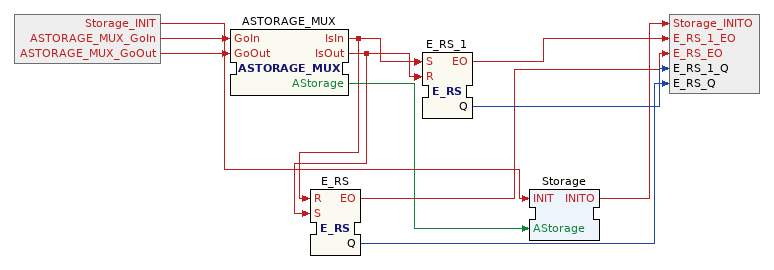
      [picture p48: application VDMA_Station1_HierarchicalControl_Distributed.StorageInternalLogicSubApp]
      FBS
        ASTORAGE_MUX : ASTORAGE_MUX;
        E_RS_1 : E_RS;
        E_RS : E_RS;
      END_FBS
      SUBAPPLICATION Storage
        EVENT_INPUT
          INIT;
        END_EVENT
        EVENT_OUTPUT
          INITO;
        END_EVENT
        SOCKETS
          AStorage : AStorage;
        END_SOCKETS
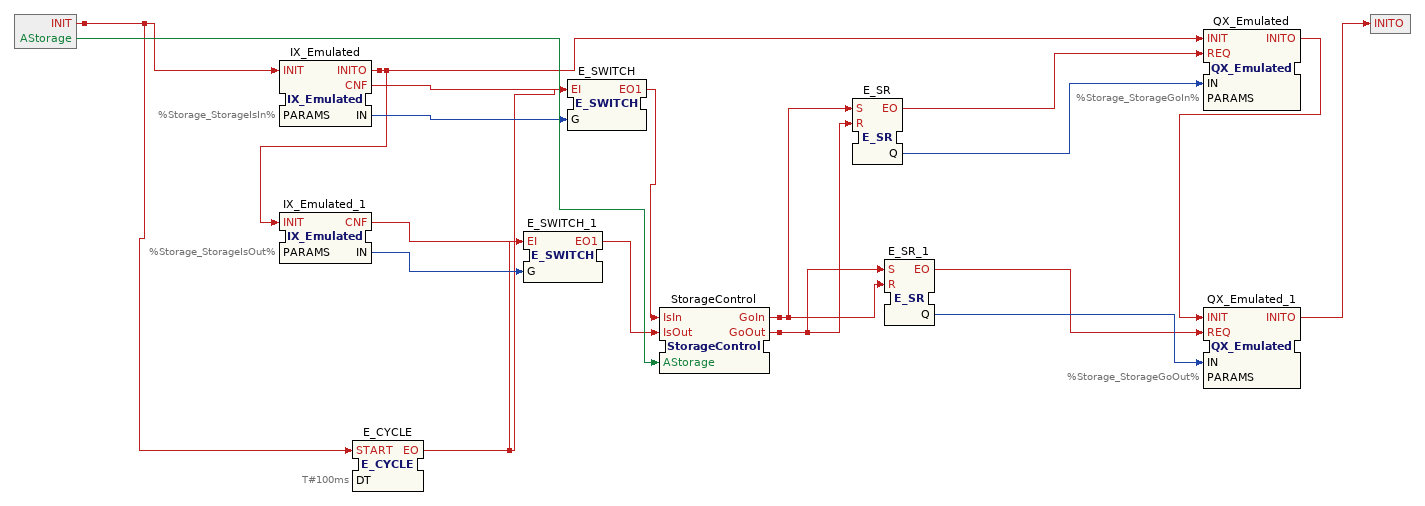
        FBS
          IX_Emulated : IX_Emulated(PARAMS := %Storage_StorageIsIn%);
          E_SWITCH : E_SWITCH;
          E_SR : E_SR;
          E_SR_1 : E_SR;
          StorageControl : StorageControl;
          E_SWITCH_1 : E_SWITCH;
          IX_Emulated_1 : IX_Emulated(PARAMS := %Storage_StorageIsOut%);
          E_CYCLE : E_CYCLE(DT := T#100ms);
          QX_Emulated_1 : QX_Emulated(PARAMS := %Storage_StorageGoOut%);
          QX_Emulated : QX_Emulated(PARAMS := %Storage_StorageGoIn%);
        END_FBS
        EVENT_CONNECTIONS
          IX_Emulated.INITO TO IX_Emulated_1.INIT;
          IX_Emulated.CNF TO E_SWITCH.EI;
          E_SWITCH.EO1 TO StorageControl.IsIn;
          StorageControl.GoIn TO E_SR.S;
          StorageControl.GoOut TO E_SR.R;
          StorageControl.GoOut TO E_SR_1.S;
          StorageControl.GoIn TO E_SR_1.R;
          E_SWITCH_1.EO1 TO StorageControl.IsOut;
          IX_Emulated_1.CNF TO E_SWITCH_1.EI;
          INIT TO IX_Emulated.INIT;
          INIT TO E_CYCLE.START;
          QX_Emulated_1.INITO TO INITO;
          IX_Emulated.INITO TO QX_Emulated.INIT;
          QX_Emulated.INITO TO QX_Emulated_1.INIT;
          E_SR.EO TO QX_Emulated.REQ;
          E_SR_1.EO TO QX_Emulated_1.REQ;
          E_CYCLE.EO TO E_SWITCH.EI;
          E_CYCLE.EO TO E_SWITCH_1.EI;
        END_CONNECTIONS
        DATA_CONNECTIONS
          IX_Emulated.IN TO E_SWITCH.G;
          IX_Emulated_1.IN TO E_SWITCH_1.G;
          E_SR.Q TO QX_Emulated.IN;
          E_SR_1.Q TO QX_Emulated_1.IN;
        END_CONNECTIONS
        ADAPTER_CONNECTIONS
          AStorage TO StorageControl.AStorage;
        END_CONNECTIONS
      END_SUBAPPLICATION
      EVENT_CONNECTIONS
        ASTORAGE_MUX.IsIn TO E_RS.R;
        ASTORAGE_MUX.IsIn TO E_RS_1.S;
        ASTORAGE_MUX.IsOut TO E_RS.S;
        ASTORAGE_MUX.IsOut TO E_RS_1.R;
        Storage_INIT TO Storage.INIT;
        Storage.INITO TO Storage_INITO;
        ASTORAGE_MUX_GoIn TO ASTORAGE_MUX.GoIn;
        ASTORAGE_MUX_GoOut TO ASTORAGE_MUX.GoOut;
        E_RS_1.EO TO E_RS_1_EO;
        E_RS.EO TO E_RS_EO;
      END_CONNECTIONS
      DATA_CONNECTIONS
        E_RS_1.Q TO E_RS_1_Q;
        E_RS.Q TO E_RS_Q;
      END_CONNECTIONS
      ADAPTER_CONNECTIONS
        ASTORAGE_MUX.AStorage TO Storage.AStorage;
      END_CONNECTIONS
    END_SUBAPPLICATION
    SUBAPPLICATION TurntableInternalLogicSubApp
      EVENT_INPUT
        ATURNTABLE_MUX_NewPosition;
        Turntable_INIT;
      END_EVENT
      EVENT_OUTPUT
        ATURNTABLE_MUX_PositionUpd;
        Turntable_INITO;
      END_EVENT
      VAR_INPUT
        ATURNTABLE_MUX_Position : WORD;
      END_VAR
      VAR_OUTPUT
        ATURNTABLE_MUX_CurrentPosition : WORD;
      END_VAR
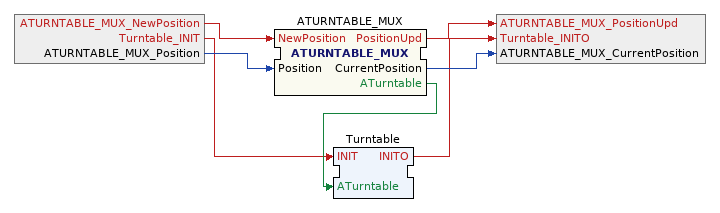
      FBS
        ATURNTABLE_MUX : ATURNTABLE_MUX;
      END_FBS
      SUBAPPLICATION Turntable
        EVENT_INPUT
          INIT;
        END_EVENT
        EVENT_OUTPUT
          INITO;
        END_EVENT
        SOCKETS
          ATurntable : ATurntable;
        END_SOCKETS
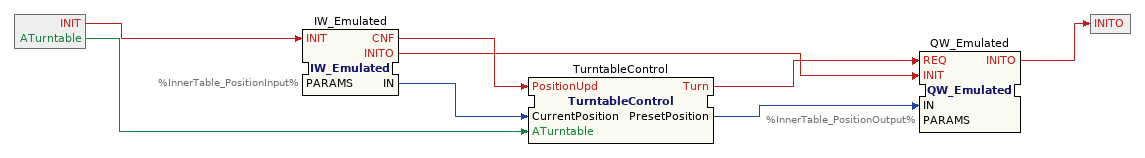
        FBS
          QW_Emulated : QW_Emulated(PARAMS := %InnerTable_PositionOutput%);
          IW_Emulated : IW_Emulated(PARAMS := %InnerTable_PositionInput%);
          TurntableControl : TurntableControl;
        END_FBS
        EVENT_CONNECTIONS
          TurntableControl.Turn TO QW_Emulated.REQ;
          IW_Emulated.CNF TO TurntableControl.PositionUpd;
          IW_Emulated.INITO TO QW_Emulated.INIT;
          INIT TO IW_Emulated.INIT;
          QW_Emulated.INITO TO INITO;
        END_CONNECTIONS
        DATA_CONNECTIONS
          TurntableControl.PresetPosition TO QW_Emulated.IN;
          IW_Emulated.IN TO TurntableControl.CurrentPosition;
        END_CONNECTIONS
        ADAPTER_CONNECTIONS
          ATurntable TO TurntableControl.ATurntable;
        END_CONNECTIONS
      END_SUBAPPLICATION
      EVENT_CONNECTIONS
        ATURNTABLE_MUX_NewPosition TO ATURNTABLE_MUX.NewPosition;
        ATURNTABLE_MUX.PositionUpd TO ATURNTABLE_MUX_PositionUpd;
        Turntable_INIT TO Turntable.INIT;
        Turntable.INITO TO Turntable_INITO;
      END_CONNECTIONS
      DATA_CONNECTIONS
        ATURNTABLE_MUX_Position TO ATURNTABLE_MUX.Position;
        ATURNTABLE_MUX.CurrentPosition TO ATURNTABLE_MUX_CurrentPosition;
      END_CONNECTIONS
      ADAPTER_CONNECTIONS
        ATURNTABLE_MUX.ATurntable TO Turntable.ATurntable;
      END_CONNECTIONS
    END_SUBAPPLICATION
    SUBAPPLICATION GripperInternalLogicSubApp
      EVENT_INPUT
        Gripper_INIT;
        AGRIPPER_MUX_Grip;
        AGRIPPER_MUX_Release;
      END_EVENT
      EVENT_OUTPUT
        E_RS_3_EO;
        Gripper_INITO;
        E_RS_2_EO;
      END_EVENT
      VAR_OUTPUT
        E_RS_3_Q : BOOL;
        E_RS_2_Q : BOOL;
      END_VAR
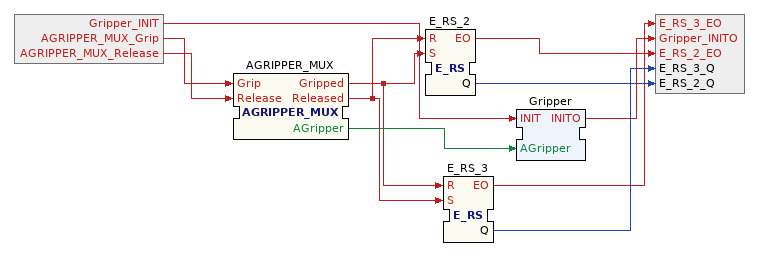
      FBS
        E_RS_3 : E_RS;
        E_RS_2 : E_RS;
        AGRIPPER_MUX : AGRIPPER_MUX;
      END_FBS
      SUBAPPLICATION Gripper
        EVENT_INPUT
          INIT;
        END_EVENT
        EVENT_OUTPUT
          INITO;
        END_EVENT
        SOCKETS
          AGripper : AGripper;
        END_SOCKETS
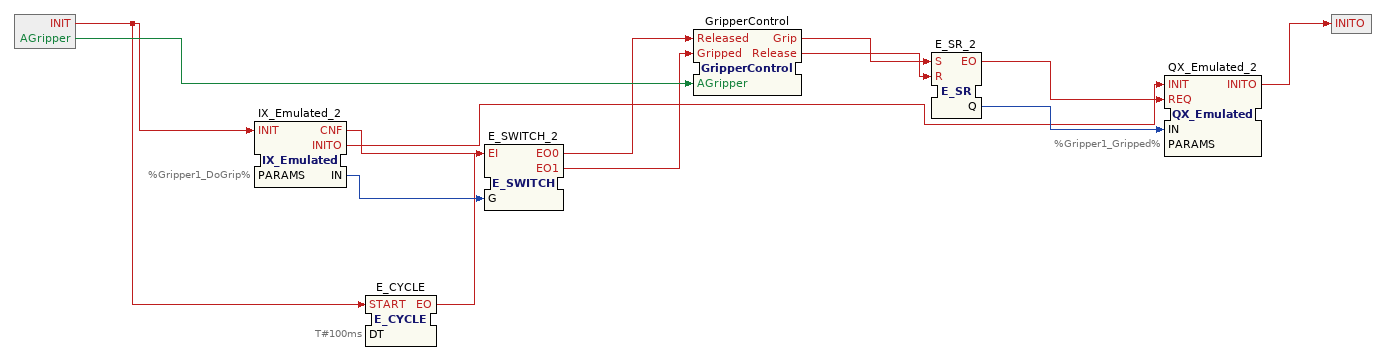
        FBS
          IX_Emulated_2 : IX_Emulated(PARAMS := %Gripper1_DoGrip%);
          E_SWITCH_2 : E_SWITCH;
          GripperControl : GripperControl;
          E_SR_2 : E_SR;
          E_CYCLE : E_CYCLE(DT := T#100ms);
          QX_Emulated_2 : QX_Emulated(PARAMS := %Gripper1_Gripped%);
        END_FBS
        EVENT_CONNECTIONS
          IX_Emulated_2.CNF TO E_SWITCH_2.EI;
          E_SWITCH_2.EO0 TO GripperControl.Released;
          E_SWITCH_2.EO1 TO GripperControl.Gripped;
          GripperControl.Grip TO E_SR_2.S;
          GripperControl.Release TO E_SR_2.R;
          E_CYCLE.EO TO E_SWITCH_2.EI;
          INIT TO E_CYCLE.START;
          INIT TO IX_Emulated_2.INIT;
          IX_Emulated_2.INITO TO QX_Emulated_2.INIT;
          QX_Emulated_2.INITO TO INITO;
          E_SR_2.EO TO QX_Emulated_2.REQ;
        END_CONNECTIONS
        DATA_CONNECTIONS
          IX_Emulated_2.IN TO E_SWITCH_2.G;
          E_SR_2.Q TO QX_Emulated_2.IN;
        END_CONNECTIONS
        ADAPTER_CONNECTIONS
          AGripper TO GripperControl.AGripper;
        END_CONNECTIONS
      END_SUBAPPLICATION
      EVENT_CONNECTIONS
        AGRIPPER_MUX.Gripped TO E_RS_3.R;
        AGRIPPER_MUX.Released TO E_RS_3.S;
        AGRIPPER_MUX.Released TO E_RS_2.R;
        AGRIPPER_MUX.Gripped TO E_RS_2.S;
        E_RS_3.EO TO E_RS_3_EO;
        Gripper_INIT TO Gripper.INIT;
        Gripper.INITO TO Gripper_INITO;
        E_RS_2.EO TO E_RS_2_EO;
        AGRIPPER_MUX_Grip TO AGRIPPER_MUX.Grip;
        AGRIPPER_MUX_Release TO AGRIPPER_MUX.Release;
      END_CONNECTIONS
      DATA_CONNECTIONS
        E_RS_3.Q TO E_RS_3_Q;
        E_RS_2.Q TO E_RS_2_Q;
      END_CONNECTIONS
      ADAPTER_CONNECTIONS
        AGRIPPER_MUX.AGripper TO Gripper.AGripper;
      END_CONNECTIONS
    END_SUBAPPLICATION
    SUBAPPLICATION RobotInternalLogicSubApp
      EVENT_INPUT
        AROBOT_MUX_PresetPositionUpd;
        Robot_INIT;
      END_EVENT
      EVENT_OUTPUT
        AROBOT_MUX_PositionUpdate;
        Robot_INITO;
      END_EVENT
      VAR_INPUT
        AROBOT_MUX_PresetPosition : WORD;
      END_VAR
      VAR_OUTPUT
        AROBOT_MUX_CurrentPosition : WORD;
      END_VAR
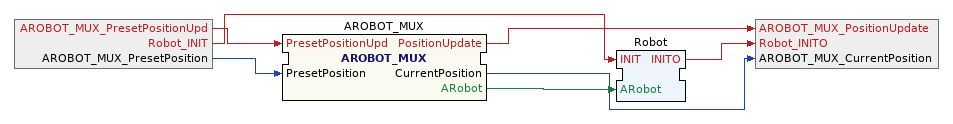
      FBS
        AROBOT_MUX : AROBOT_MUX;
      END_FBS
      SUBAPPLICATION Robot
        EVENT_INPUT
          INIT;
        END_EVENT
        EVENT_OUTPUT
          INITO;
        END_EVENT
        SOCKETS
          ARobot : ARobot;
        END_SOCKETS
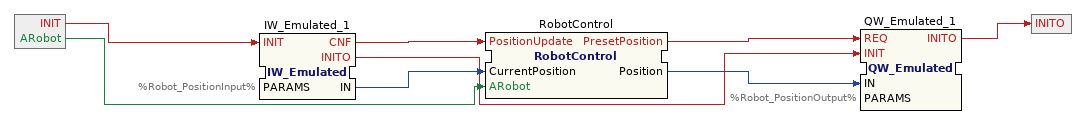
        FBS
          IW_Emulated_1 : IW_Emulated(PARAMS := %Robot_PositionInput%);
          RobotControl : RobotControl;
          QW_Emulated_1 : QW_Emulated(PARAMS := %Robot_PositionOutput%);
        END_FBS
        EVENT_CONNECTIONS
          IW_Emulated_1.CNF TO RobotControl.PositionUpdate;
          RobotControl.PresetPosition TO QW_Emulated_1.REQ;
          IW_Emulated_1.INITO TO QW_Emulated_1.INIT;
          QW_Emulated_1.INITO TO INITO;
          INIT TO IW_Emulated_1.INIT;
        END_CONNECTIONS
        DATA_CONNECTIONS
          IW_Emulated_1.IN TO RobotControl.CurrentPosition;
          RobotControl.Position TO QW_Emulated_1.IN;
        END_CONNECTIONS
        ADAPTER_CONNECTIONS
          ARobot TO RobotControl.ARobot;
        END_CONNECTIONS
      END_SUBAPPLICATION
      EVENT_CONNECTIONS
        AROBOT_MUX_PresetPositionUpd TO AROBOT_MUX.PresetPositionUpd;
        AROBOT_MUX.PositionUpdate TO AROBOT_MUX_PositionUpdate;
        Robot_INIT TO Robot.INIT;
        Robot.INITO TO Robot_INITO;
      END_CONNECTIONS
      DATA_CONNECTIONS
        AROBOT_MUX_PresetPosition TO AROBOT_MUX.PresetPosition;
        AROBOT_MUX.CurrentPosition TO AROBOT_MUX_CurrentPosition;
      END_CONNECTIONS
      ADAPTER_CONNECTIONS
        AROBOT_MUX.ARobot TO Robot.ARobot;
      END_CONNECTIONS
    END_SUBAPPLICATION
    EVENT_CONNECTIONS
      SERVER_0.IND TO SERVER_0.RSP;
      SERVER_1.IND TO SERVER_1.RSP;
      SERVER_0.INITO TO SERVER_1.INIT;
      SERVER_5.IND TO SERVER_5.RSP;
      SERVER_4.IND TO SERVER_4.RSP;
      SERVER_4.INITO TO SERVER_5.INIT;
      CLIENT_4.INITO TO CLIENT_5.INIT;
      CLIENT_0.INITO TO CLIENT_3.INIT;
      SUBSCRIBE_2.IND TO TurntableSubApp.PositionUpd;
      SUBSCRIBE_1.IND TO RobotSubApp.PositionUpdate;
      SERVER_5.INITO TO PUBLISH_5.INIT;
      PUBLISH_5.INITO TO PUBLISH_4.INIT;
      SUBSCRIBE_3.INITO TO CLIENT_0.INIT;
      SERVER_1.INITO TO PUBLISH_0.INIT;
      PUBLISH_0.INITO TO PUBLISH_1.INIT;
      SUBSCRIBE_2.INITO TO SUBSCRIBE_4.INIT;
      SUBSCRIBE_4.INITO TO SUBSCRIBE_5.INIT;
      SUBSCRIBE_5.INITO TO CLIENT_4.INIT;
      SUBSCRIBE_5.INITO TO SUBSCRIBE_1.INIT;
      SUBSCRIBE_9.INITO TO SUBSCRIBE_3.INIT;
      CLIENT_3.INITO TO SUBSCRIBE_2.INIT;
      SERVER_3.IND TO SERVER_3.RSP;
      SERVER_3.INITO TO PUBLISH_3.INIT;
      SUBSCRIBE_2.INITO TO CLIENT_2.INIT;
      TurntableSubApp.NewPosition TO CLIENT_2.REQ;
      SUBSCRIBE_1.INITO TO CLIENT_1.INIT;
      RobotSubApp.PresetPositionUpd TO CLIENT_1.REQ;
      SERVER_2.IND TO SERVER_2.RSP;
      SERVER_2.INITO TO PUBLISH_2.INIT;
      SUBSCRIBE_9.IND TO StorageSubApp.E_SWITCH_1_EI;
      SUBSCRIBE_3.IND TO StorageSubApp.E_SWITCH_EI;
      StorageSubApp.ASTORAGE_DEMUX_GoIn TO CLIENT_0.REQ;
      StorageSubApp.ASTORAGE_DEMUX_GoOut TO CLIENT_3.REQ;
      SUBSCRIBE_4.IND TO GripperSubApp.E_SWITCH_2_EI;
      GripperSubApp.AGRIPPER_DEMUX_Grip TO CLIENT_4.REQ;
      GripperSubApp.AGRIPPER_DEMUX_Release TO CLIENT_5.REQ;
      SUBSCRIBE_5.IND TO GripperSubApp.E_SWITCH_3_EI;
      SERVER_5.INITO TO StorageInternalLogicSubApp.Storage_INIT;
      SERVER_4.IND TO StorageInternalLogicSubApp.ASTORAGE_MUX_GoIn;
      SERVER_5.IND TO StorageInternalLogicSubApp.ASTORAGE_MUX_GoOut;
      StorageInternalLogicSubApp.E_RS_1_EO TO PUBLISH_5.REQ;
      StorageInternalLogicSubApp.E_RS_EO TO PUBLISH_4.REQ;
      SERVER_3.IND TO TurntableInternalLogicSubApp.ATURNTABLE_MUX_NewPosition;
      TurntableInternalLogicSubApp.ATURNTABLE_MUX_PositionUpd TO PUBLISH_3.REQ;
      StorageInternalLogicSubApp.Storage_INITO TO TurntableInternalLogicSubApp.Turntable_INIT;
      TurntableInternalLogicSubApp.Turntable_INITO TO SERVER_3.INIT;
      GripperInternalLogicSubApp.E_RS_3_EO TO PUBLISH_1.REQ;
      TurntableInternalLogicSubApp.Turntable_INITO TO GripperInternalLogicSubApp.Gripper_INIT;
      GripperInternalLogicSubApp.Gripper_INITO TO SERVER_0.INIT;
      GripperInternalLogicSubApp.E_RS_2_EO TO PUBLISH_0.REQ;
      SERVER_0.IND TO GripperInternalLogicSubApp.AGRIPPER_MUX_Grip;
      SERVER_1.IND TO GripperInternalLogicSubApp.AGRIPPER_MUX_Release;
      SERVER_2.IND TO RobotInternalLogicSubApp.AROBOT_MUX_PresetPositionUpd;
      RobotInternalLogicSubApp.AROBOT_MUX_PositionUpdate TO PUBLISH_2.REQ;
      GripperInternalLogicSubApp.Gripper_INITO TO RobotInternalLogicSubApp.Robot_INIT;
      RobotInternalLogicSubApp.Robot_INITO TO SERVER_2.INIT;
    END_CONNECTIONS
    DATA_CONNECTIONS
      SUBSCRIBE_1.RD_1 TO RobotSubApp.CurrentPosition;
      SUBSCRIBE_2.RD_1 TO TurntableSubApp.CurrentPosition;
      TurntableSubApp.Position TO CLIENT_2.SD_1;
      RobotSubApp.PresetPosition TO CLIENT_1.SD_1;
      SUBSCRIBE_9.RD_1 TO StorageSubApp.E_SWITCH_1_G;
      SUBSCRIBE_3.RD_1 TO StorageSubApp.E_SWITCH_G;
      SUBSCRIBE_4.RD_1 TO GripperSubApp.E_SWITCH_2_G;
      SUBSCRIBE_5.RD_1 TO GripperSubApp.E_SWITCH_3_G;
      StorageInternalLogicSubApp.E_RS_1_Q TO PUBLISH_5.SD_1;
      StorageInternalLogicSubApp.E_RS_Q TO PUBLISH_4.SD_1;
      SERVER_3.RD_1 TO TurntableInternalLogicSubApp.ATURNTABLE_MUX_Position;
      TurntableInternalLogicSubApp.ATURNTABLE_MUX_CurrentPosition TO PUBLISH_3.SD_1;
      GripperInternalLogicSubApp.E_RS_3_Q TO PUBLISH_1.SD_1;
      GripperInternalLogicSubApp.E_RS_2_Q TO PUBLISH_0.SD_1;
      SERVER_2.RD_1 TO RobotInternalLogicSubApp.AROBOT_MUX_PresetPosition;
      RobotInternalLogicSubApp.AROBOT_MUX_CurrentPosition TO PUBLISH_2.SD_1;
    END_CONNECTIONS
    ADAPTER_CONNECTIONS
      Station1Control.ADepot TO DepotControl.ADepot;
      Station1Control.AHandling TO HandlingControl.AHandling;
      HandlingControl.ARobot TO RobotSubApp.ARobot;
      DepotControl.ATurntable TO TurntableSubApp.ATurntable;
      DepotControl.AStorage TO StorageSubApp.ASTORAGE_DEMUX_AStorage;
      HandlingControl.AGripper TO GripperSubApp.AGRIPPER_DEMUX_AGripper;
    END_CONNECTIONS
  END_APPLICATION
  APPLICATION VDMA_Station1_SkillbasedControl_Distributed
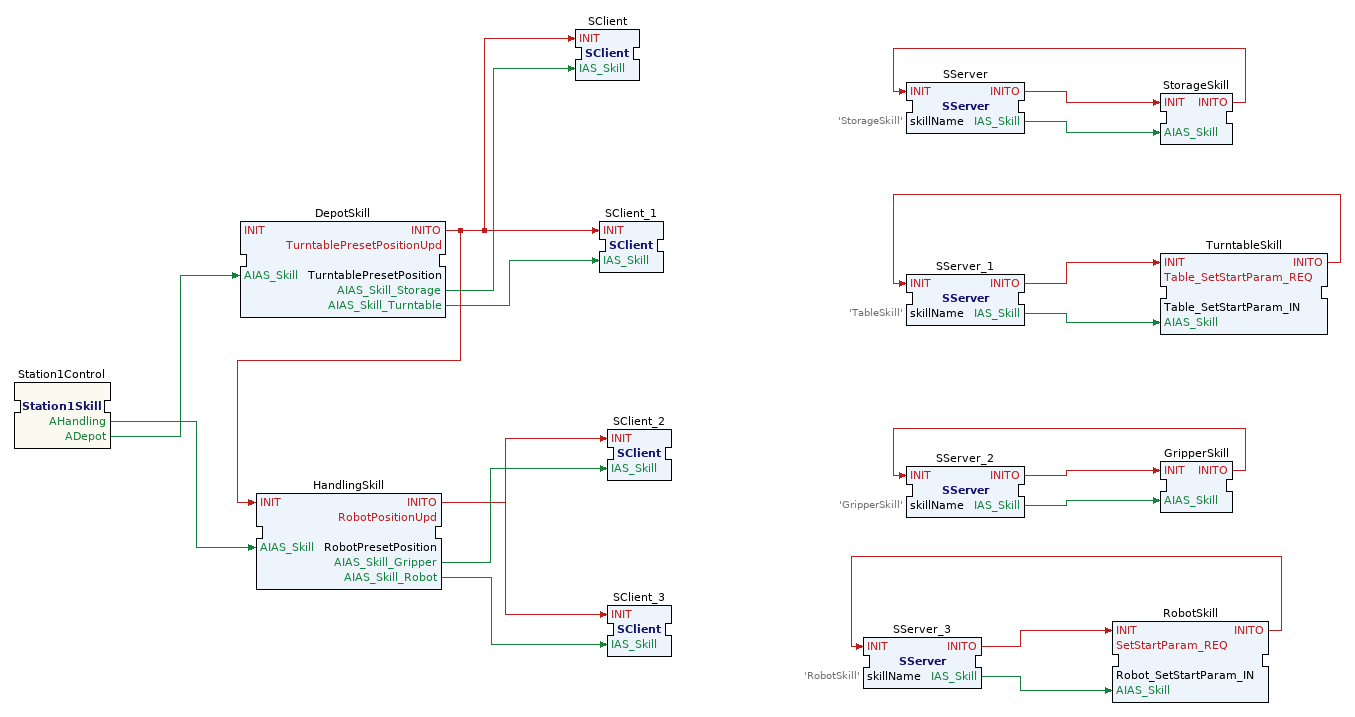
    FBS
      Station1Control : Station1Skill;
    END_FBS
    SUBAPPS
      SClient : SClient;
      SClient_1 : SClient;
      SClient_2 : SClient;
      SClient_3 : SClient;
      SServer : SServer(skillName := 'StorageSkill');
      SServer_1 : SServer(skillName := 'TableSkill');
      SServer_2 : SServer(skillName := 'GripperSkill');
      SServer_3 : SServer(skillName := 'RobotSkill');
    END_SUBAPPS
    SUBAPPLICATION StorageSkill
      EVENT_INPUT
        INIT;
      END_EVENT
      EVENT_OUTPUT
        INITO;
      END_EVENT
      SOCKETS
        AIAS_Skill : IAS_Skill;
      END_SOCKETS
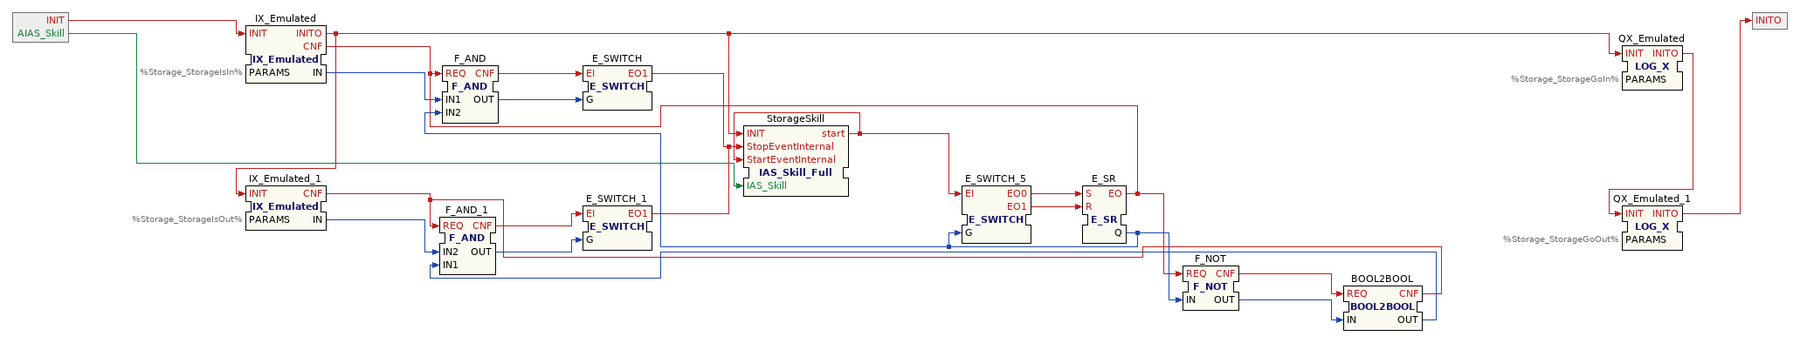
      FBS
        E_SWITCH_5 : E_SWITCH;
        IX_Emulated : IX_Emulated(PARAMS := %Storage_StorageIsIn%);
        QX_Emulated_1 : LOG_X(PARAMS := %Storage_StorageGoOut%);
        F_NOT : F_NOT;
        QX_Emulated : LOG_X(PARAMS := %Storage_StorageGoIn%);
        IX_Emulated_1 : IX_Emulated(PARAMS := %Storage_StorageIsOut%);
        E_SWITCH : E_SWITCH;
        E_SWITCH_1 : E_SWITCH;
        StorageSkill : IAS_Skill_Full;
        F_AND : F_AND;
        BOOL2BOOL : BOOL2BOOL;
        F_AND_1 : F_AND;
        E_SR : E_SR;
      END_FBS
      EVENT_CONNECTIONS
        StorageSkill.start TO E_SWITCH_5.EI;
        E_SWITCH_5.EO0 TO E_SR.S;
        E_SWITCH_5.EO1 TO E_SR.R;
        IX_Emulated.INITO TO IX_Emulated_1.INIT;
        IX_Emulated.INITO TO QX_Emulated.INIT;
        IX_Emulated.INITO TO StorageSkill.INIT;
        IX_Emulated.CNF TO F_AND.REQ;
        QX_Emulated.INITO TO QX_Emulated_1.INIT;
        E_SR.EO TO F_NOT.REQ;
        F_NOT.CNF TO BOOL2BOOL.REQ;
        IX_Emulated_1.CNF TO F_AND_1.REQ;
        F_AND.CNF TO E_SWITCH.EI;
        E_SWITCH.EO1 TO StorageSkill.StopEventInternal;
        F_AND_1.CNF TO E_SWITCH_1.EI;
        E_SWITCH_1.EO1 TO StorageSkill.StopEventInternal;
        StorageSkill.start TO StorageSkill.StartEventInternal;
        E_SR.EO TO F_AND.REQ;
        BOOL2BOOL.CNF TO F_AND_1.REQ;
        INIT TO IX_Emulated.INIT;
        QX_Emulated_1.INITO TO INITO;
      END_CONNECTIONS
      DATA_CONNECTIONS
        E_SR.Q TO E_SWITCH_5.G;
        IX_Emulated.IN TO F_AND.IN1;
        E_SR.Q TO F_NOT.IN;
        F_NOT.OUT TO BOOL2BOOL.IN;
        IX_Emulated_1.IN TO F_AND_1.IN2;
        F_AND.OUT TO E_SWITCH.G;
        F_AND_1.OUT TO E_SWITCH_1.G;
        E_SR.Q TO F_AND.IN2;
        BOOL2BOOL.OUT TO F_AND_1.IN1;
      END_CONNECTIONS
      ADAPTER_CONNECTIONS
        AIAS_Skill TO StorageSkill.IAS_Skill;
      END_CONNECTIONS
    END_SUBAPPLICATION
    SUBAPPLICATION TurntableSkill
      EVENT_INPUT
        INIT;
        Table_SetStartParam_REQ;
      END_EVENT
      EVENT_OUTPUT
        INITO;
      END_EVENT
      VAR_INPUT
        Table_SetStartParam_IN : WORD;
      END_VAR
      SOCKETS
        AIAS_Skill : IAS_Skill;
      END_SOCKETS
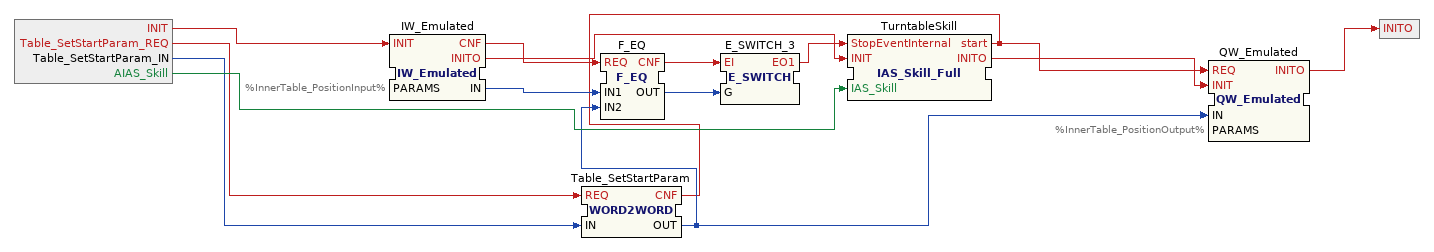
      FBS
        F_EQ : F_EQ;
        E_SWITCH_3 : E_SWITCH;
        Table_SetStartParam : WORD2WORD;
        QW_Emulated : QW_Emulated(PARAMS := %InnerTable_PositionOutput%);
        TurntableSkill : IAS_Skill_Full;
        IW_Emulated : IW_Emulated(PARAMS := %InnerTable_PositionInput%);
      END_FBS
      EVENT_CONNECTIONS
        IW_Emulated.CNF TO F_EQ.REQ;
        TurntableSkill.start TO F_EQ.REQ;
        Table_SetStartParam.CNF TO F_EQ.REQ;
        F_EQ.CNF TO E_SWITCH_3.EI;
        E_SWITCH_3.EO1 TO TurntableSkill.StopEventInternal;
        TurntableSkill.start TO QW_Emulated.REQ;
        Table_SetStartParam_REQ TO Table_SetStartParam.REQ;
        INIT TO IW_Emulated.INIT;
        IW_Emulated.INITO TO TurntableSkill.INIT;
        TurntableSkill.INITO TO QW_Emulated.INIT;
        QW_Emulated.INITO TO INITO;
      END_CONNECTIONS
      DATA_CONNECTIONS
        IW_Emulated.IN TO F_EQ.IN1;
        Table_SetStartParam.OUT TO F_EQ.IN2;
        F_EQ.OUT TO E_SWITCH_3.G;
        Table_SetStartParam.OUT TO QW_Emulated.IN;
        Table_SetStartParam_IN TO Table_SetStartParam.IN;
      END_CONNECTIONS
      ADAPTER_CONNECTIONS
        AIAS_Skill TO TurntableSkill.IAS_Skill;
      END_CONNECTIONS
    END_SUBAPPLICATION
    SUBAPPLICATION DepotSkill
      EVENT_INPUT
        INIT;
      END_EVENT
      EVENT_OUTPUT
        INITO;
        TurntablePresetPositionUpd;
      END_EVENT
      VAR_OUTPUT
        TurntablePresetPosition : WORD;
      END_VAR
      SOCKETS
        AIAS_Skill : IAS_Skill;
      END_SOCKETS
      PLUGS
        AIAS_Skill_Storage : IAS_Skill;
        AIAS_Skill_Turntable : IAS_Skill;
      END_PLUGS
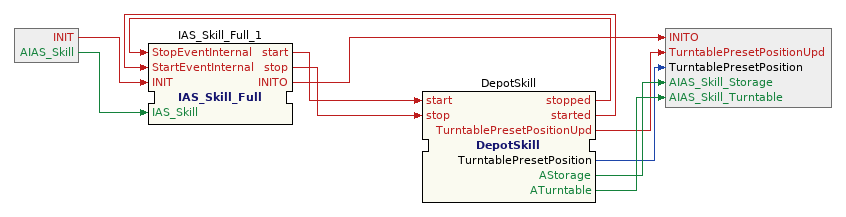
      FBS
        IAS_Skill_Full_1 : IAS_Skill_Full;
        DepotSkill : DepotSkill;
      END_FBS
      EVENT_CONNECTIONS
        DepotSkill.stopped TO IAS_Skill_Full_1.StopEventInternal;
        DepotSkill.started TO IAS_Skill_Full_1.StartEventInternal;
        IAS_Skill_Full_1.start TO DepotSkill.start;
        IAS_Skill_Full_1.stop TO DepotSkill.stop;
        DepotSkill.TurntablePresetPositionUpd TO TurntablePresetPositionUpd;
        INIT TO IAS_Skill_Full_1.INIT;
        IAS_Skill_Full_1.INITO TO INITO;
      END_CONNECTIONS
      DATA_CONNECTIONS
        DepotSkill.TurntablePresetPosition TO TurntablePresetPosition;
      END_CONNECTIONS
      ADAPTER_CONNECTIONS
        AIAS_Skill TO IAS_Skill_Full_1.IAS_Skill;
        DepotSkill.AStorage TO AIAS_Skill_Storage;
        DepotSkill.ATurntable TO AIAS_Skill_Turntable;
      END_CONNECTIONS
    END_SUBAPPLICATION
    SUBAPPLICATION GripperSkill
      EVENT_INPUT
        INIT;
      END_EVENT
      EVENT_OUTPUT
        INITO;
      END_EVENT
      SOCKETS
        AIAS_Skill : IAS_Skill;
      END_SOCKETS
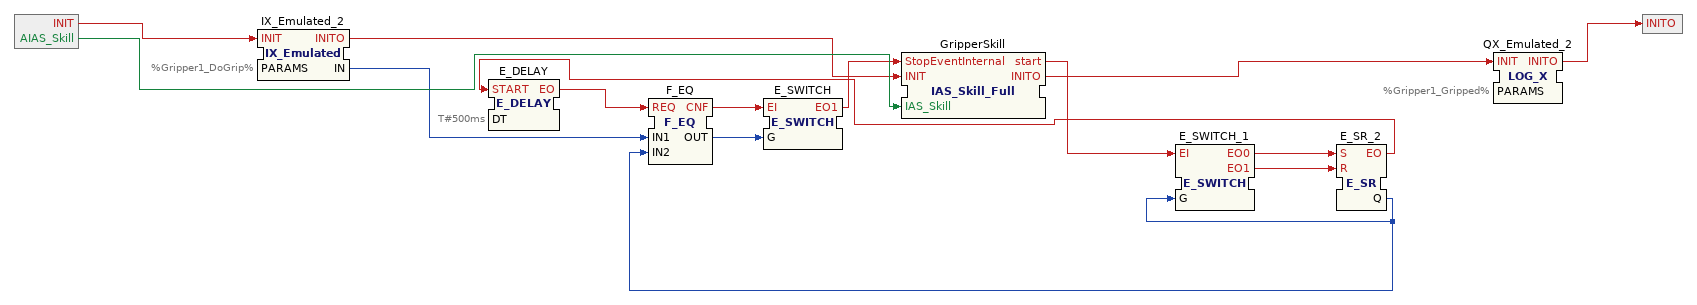
      FBS
        GripperSkill : IAS_Skill_Full;
        F_EQ : F_EQ;
        E_SWITCH_1 : E_SWITCH;
        IX_Emulated_2 : IX_Emulated(PARAMS := %Gripper1_DoGrip%);
        QX_Emulated_2 : LOG_X(PARAMS := %Gripper1_Gripped%);
        E_DELAY : E_DELAY(DT := T#500ms);
        E_SWITCH : E_SWITCH;
        E_SR_2 : E_SR;
      END_FBS
      EVENT_CONNECTIONS
        E_SWITCH.EO1 TO GripperSkill.StopEventInternal;
        GripperSkill.start TO E_SWITCH_1.EI;
        E_DELAY.EO TO F_EQ.REQ;
        F_EQ.CNF TO E_SWITCH.EI;
        E_SWITCH_1.EO0 TO E_SR_2.S;
        E_SWITCH_1.EO1 TO E_SR_2.R;
        E_SR_2.EO TO E_DELAY.START;
        INIT TO IX_Emulated_2.INIT;
        IX_Emulated_2.INITO TO GripperSkill.INIT;
        GripperSkill.INITO TO QX_Emulated_2.INIT;
        QX_Emulated_2.INITO TO INITO;
      END_CONNECTIONS
      DATA_CONNECTIONS
        IX_Emulated_2.IN TO F_EQ.IN1;
        E_SR_2.Q TO F_EQ.IN2;
        F_EQ.OUT TO E_SWITCH.G;
        E_SR_2.Q TO E_SWITCH_1.G;
      END_CONNECTIONS
      ADAPTER_CONNECTIONS
        AIAS_Skill TO GripperSkill.IAS_Skill;
      END_CONNECTIONS
    END_SUBAPPLICATION
    SUBAPPLICATION RobotSkill
      EVENT_INPUT
        INIT;
        SetStartParam_REQ;
      END_EVENT
      EVENT_OUTPUT
        INITO;
      END_EVENT
      VAR_INPUT
        Robot_SetStartParam_IN : WORD;
      END_VAR
      SOCKETS
        AIAS_Skill : IAS_Skill;
      END_SOCKETS
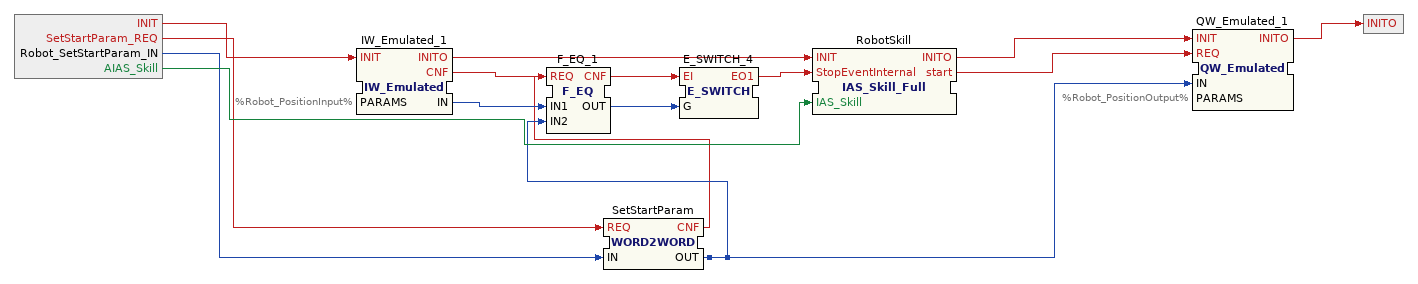
      FBS
        RobotSkill : IAS_Skill_Full;
        IW_Emulated_1 : IW_Emulated(PARAMS := %Robot_PositionInput%);
        E_SWITCH_4 : E_SWITCH;
        F_EQ_1 : F_EQ;
        QW_Emulated_1 : QW_Emulated(PARAMS := %Robot_PositionOutput%);
        SetStartParam : WORD2WORD;
      END_FBS
      EVENT_CONNECTIONS
        IW_Emulated_1.INITO TO RobotSkill.INIT;
        E_SWITCH_4.EO1 TO RobotSkill.StopEventInternal;
        RobotSkill.INITO TO QW_Emulated_1.INIT;
        RobotSkill.start TO QW_Emulated_1.REQ;
        IW_Emulated_1.CNF TO F_EQ_1.REQ;
        F_EQ_1.CNF TO E_SWITCH_4.EI;
        SetStartParam.CNF TO F_EQ_1.REQ;
        INIT TO IW_Emulated_1.INIT;
        SetStartParam_REQ TO SetStartParam.REQ;
        QW_Emulated_1.INITO TO INITO;
      END_CONNECTIONS
      DATA_CONNECTIONS
        IW_Emulated_1.IN TO F_EQ_1.IN1;
        F_EQ_1.OUT TO E_SWITCH_4.G;
        SetStartParam.OUT TO F_EQ_1.IN2;
        SetStartParam.OUT TO QW_Emulated_1.IN;
        Robot_SetStartParam_IN TO SetStartParam.IN;
      END_CONNECTIONS
      ADAPTER_CONNECTIONS
        AIAS_Skill TO RobotSkill.IAS_Skill;
      END_CONNECTIONS
    END_SUBAPPLICATION
    SUBAPPLICATION HandlingSkill
      EVENT_INPUT
        INIT;
      END_EVENT
      EVENT_OUTPUT
        INITO;
        RobotPositionUpd;
      END_EVENT
      VAR_OUTPUT
        RobotPresetPosition : WORD;
      END_VAR
      SOCKETS
        AIAS_Skill : IAS_Skill;
      END_SOCKETS
      PLUGS
        AIAS_Skill_Gripper : IAS_Skill;
        AIAS_Skill_Robot : IAS_Skill;
      END_PLUGS
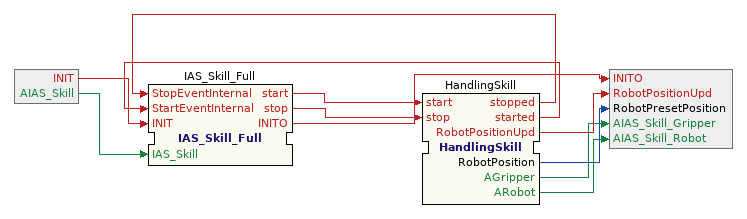
      FBS
        IAS_Skill_Full : IAS_Skill_Full;
        HandlingSkill : HandlingSkill;
      END_FBS
      EVENT_CONNECTIONS
        HandlingSkill.stopped TO IAS_Skill_Full.StopEventInternal;
        HandlingSkill.started TO IAS_Skill_Full.StartEventInternal;
        IAS_Skill_Full.start TO HandlingSkill.start;
        IAS_Skill_Full.stop TO HandlingSkill.stop;
        HandlingSkill.RobotPositionUpd TO RobotPositionUpd;
        INIT TO IAS_Skill_Full.INIT;
        IAS_Skill_Full.INITO TO INITO;
      END_CONNECTIONS
      DATA_CONNECTIONS
        HandlingSkill.RobotPosition TO RobotPresetPosition;
      END_CONNECTIONS
      ADAPTER_CONNECTIONS
        AIAS_Skill TO IAS_Skill_Full.IAS_Skill;
        HandlingSkill.AGripper TO AIAS_Skill_Gripper;
        HandlingSkill.ARobot TO AIAS_Skill_Robot;
      END_CONNECTIONS
    END_SUBAPPLICATION
    EVENT_CONNECTIONS
      DepotSkill.INITO TO HandlingSkill.INIT;
      HandlingSkill.INITO TO SClient_3.INIT;
      HandlingSkill.INITO TO SClient_2.INIT;
      DepotSkill.INITO TO SClient_1.INIT;
      DepotSkill.INITO TO SClient.INIT;
      SServer.INITO TO StorageSkill.INIT;
      StorageSkill.INITO TO SServer.INIT;
      SServer_1.INITO TO TurntableSkill.INIT;
      TurntableSkill.INITO TO SServer_1.INIT;
      SServer_2.INITO TO GripperSkill.INIT;
      GripperSkill.INITO TO SServer_2.INIT;
      SServer_3.INITO TO RobotSkill.INIT;
      RobotSkill.INITO TO SServer_3.INIT;
    END_CONNECTIONS
    ADAPTER_CONNECTIONS
      Station1Control.AHandling TO HandlingSkill.AIAS_Skill;
      Station1Control.ADepot TO DepotSkill.AIAS_Skill;
      DepotSkill.AIAS_Skill_Storage TO SClient.IAS_Skill;
      DepotSkill.AIAS_Skill_Turntable TO SClient_1.IAS_Skill;
      HandlingSkill.AIAS_Skill_Gripper TO SClient_2.IAS_Skill;
      HandlingSkill.AIAS_Skill_Robot TO SClient_3.IAS_Skill;
      SServer.IAS_Skill TO StorageSkill.AIAS_Skill;
      SServer_1.IAS_Skill TO TurntableSkill.AIAS_Skill;
      SServer_2.IAS_Skill TO GripperSkill.AIAS_Skill;
      SServer_3.IAS_Skill TO RobotSkill.AIAS_Skill;
    END_CONNECTIONS
  END_APPLICATION
  APPLICATION VDMA_Station1_EmulatorApp_SingleDevice
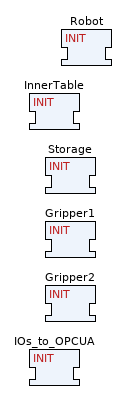
    SUBAPPLICATION Robot
      EVENT_INPUT
        INIT;
      END_EVENT
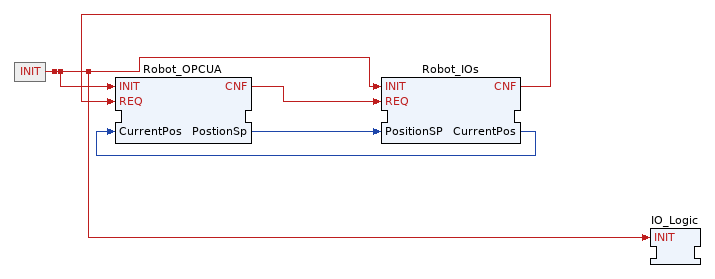
      SUBAPPLICATION IO_Logic
        EVENT_INPUT
          INIT;
        END_EVENT
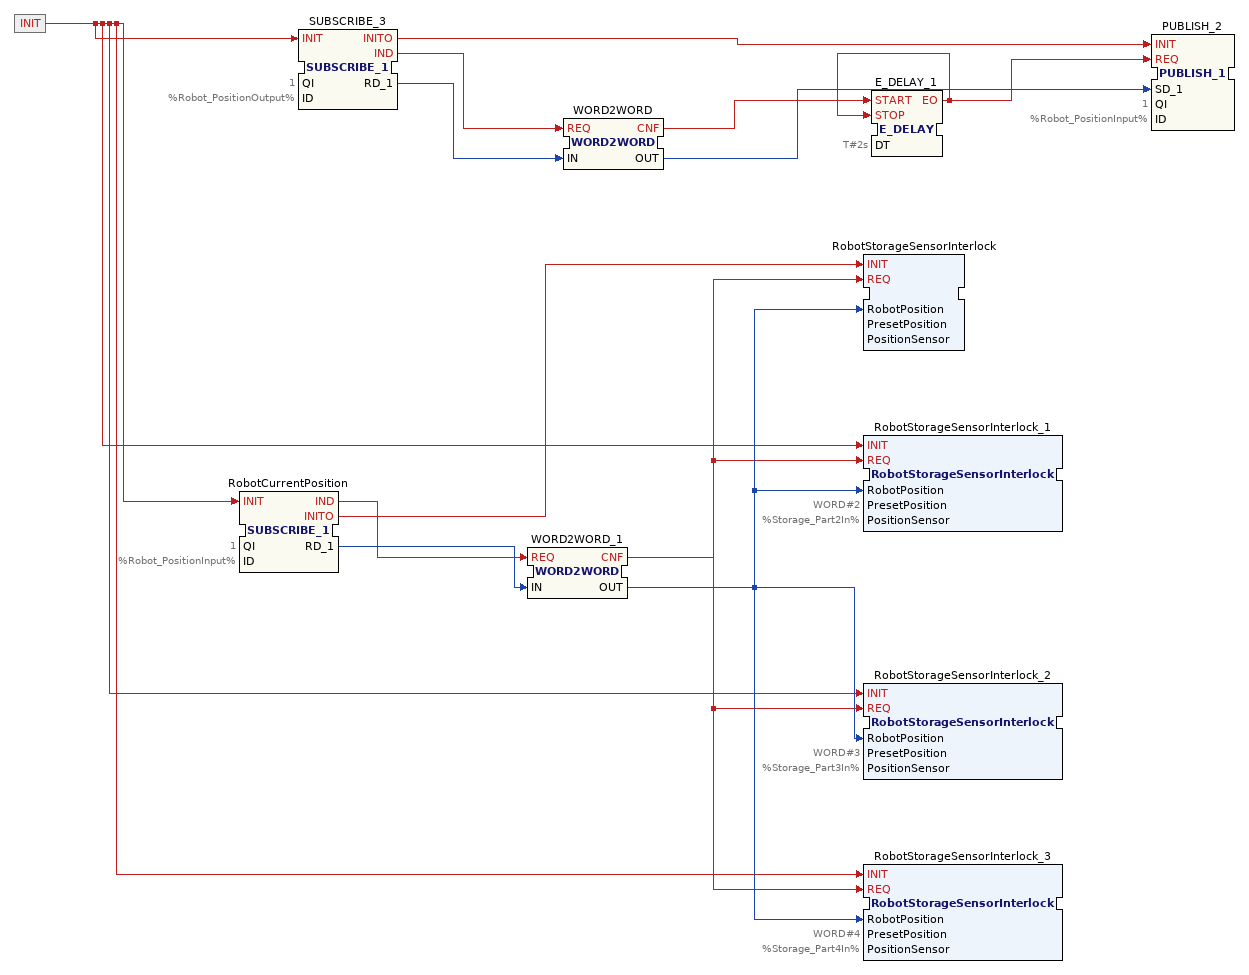
        FBS
          SUBSCRIBE_3 : SUBSCRIBE_1(QI := 1, ID := %Robot_PositionOutput%);
          WORD2WORD : WORD2WORD;
          E_DELAY_1 : E_DELAY(DT := T#2s);
          PUBLISH_2 : PUBLISH_1(QI := 1, ID := %Robot_PositionInput%);
          RobotCurrentPosition : SUBSCRIBE_1(QI := 1, ID := %Robot_PositionInput%);
          WORD2WORD_1 : WORD2WORD;
        END_FBS
        SUBAPPS
          RobotStorageSensorInterlock_1 : RobotStorageSensorInterlock(PresetPosition := WORD#2, PositionSensor := %Storage_Part2In%);
          RobotStorageSensorInterlock_2 : RobotStorageSensorInterlock(PresetPosition := WORD#3, PositionSensor := %Storage_Part3In%);
          RobotStorageSensorInterlock_3 : RobotStorageSensorInterlock(PresetPosition := WORD#4, PositionSensor := %Storage_Part4In%);
        END_SUBAPPS
        SUBAPPLICATION RobotStorageSensorInterlock
          EVENT_INPUT
            INIT;
            REQ;
          END_EVENT
          VAR_INPUT
            RobotPosition : ANY_ELEMENTARY;
            PresetPosition : WORD := WORD#1;
            PositionSensor : WSTRING := %Storage_Part1In%;
          END_VAR
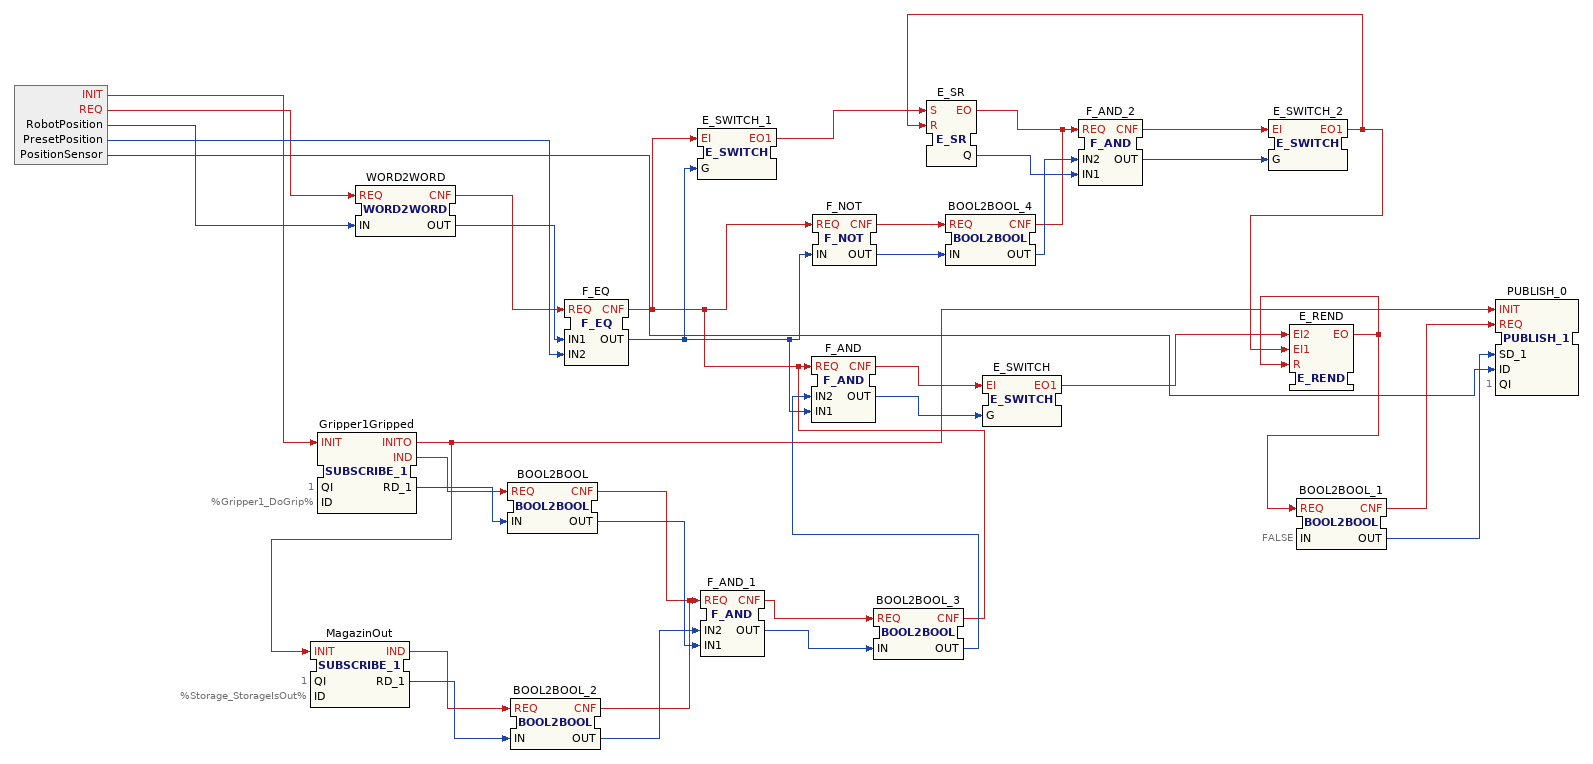
          FBS
            E_SWITCH : E_SWITCH;
            MagazinOut : SUBSCRIBE_1(QI := 1, ID := %Storage_StorageIsOut%);
            BOOL2BOOL : BOOL2BOOL;
            BOOL2BOOL_3 : BOOL2BOOL;
            Gripper1Gripped : SUBSCRIBE_1(QI := 1, ID := %Gripper1_DoGrip%);
            BOOL2BOOL_1 : BOOL2BOOL(IN := FALSE);
            F_EQ : F_EQ;
            BOOL2BOOL_2 : BOOL2BOOL;
            F_AND_1 : F_AND;
            F_AND : F_AND;
            E_REND : E_REND;
            PUBLISH_0 : PUBLISH_1(QI := 1);
            E_SR : E_SR;
            E_SWITCH_1 : E_SWITCH;
            F_AND_2 : F_AND;
            E_SWITCH_2 : E_SWITCH;
            F_NOT : F_NOT;
            BOOL2BOOL_4 : BOOL2BOOL;
            WORD2WORD : WORD2WORD;
          END_FBS
          EVENT_CONNECTIONS
            F_NOT.CNF TO BOOL2BOOL_4.REQ;
            F_EQ.CNF TO E_SWITCH_1.EI;
            Gripper1Gripped.INITO TO PUBLISH_0.INIT;
            MagazinOut.IND TO BOOL2BOOL_2.REQ;
            E_SR.EO TO F_AND_2.REQ;
            E_SWITCH_1.EO1 TO E_SR.S;
            F_AND.CNF TO E_SWITCH.EI;
            E_SWITCH.EO1 TO E_REND.EI2;
            BOOL2BOOL_4.CNF TO F_AND_2.REQ;
            BOOL2BOOL.CNF TO F_AND_1.REQ;
            Gripper1Gripped.INITO TO MagazinOut.INIT;
            Gripper1Gripped.IND TO BOOL2BOOL.REQ;
            F_EQ.CNF TO F_AND.REQ;
            BOOL2BOOL_1.CNF TO PUBLISH_0.REQ;
            E_REND.EO TO BOOL2BOOL_1.REQ;
            F_AND_2.CNF TO E_SWITCH_2.EI;
            E_SWITCH_2.EO1 TO E_REND.EI1;
            BOOL2BOOL_3.CNF TO F_AND.REQ;
            E_SWITCH_2.EO1 TO E_SR.R;
            F_AND_1.CNF TO BOOL2BOOL_3.REQ;
            E_REND.EO TO E_REND.R;
            BOOL2BOOL_2.CNF TO F_AND_1.REQ;
            F_EQ.CNF TO F_NOT.REQ;
            INIT TO Gripper1Gripped.INIT;
            REQ TO WORD2WORD.REQ;
            WORD2WORD.CNF TO F_EQ.REQ;
          END_CONNECTIONS
          DATA_CONNECTIONS
            F_EQ.OUT TO E_SWITCH_1.G;
            BOOL2BOOL_2.OUT TO F_AND_1.IN2;
            BOOL2BOOL_4.OUT TO F_AND_2.IN2;
            E_SR.Q TO F_AND_2.IN1;
            F_EQ.OUT TO F_NOT.IN;
            BOOL2BOOL_1.OUT TO PUBLISH_0.SD_1;
            F_AND.OUT TO E_SWITCH.G;
            BOOL2BOOL.OUT TO F_AND_1.IN1;
            F_NOT.OUT TO BOOL2BOOL_4.IN;
            Gripper1Gripped.RD_1 TO BOOL2BOOL.IN;
            BOOL2BOOL_3.OUT TO F_AND.IN2;
            F_EQ.OUT TO F_AND.IN1;
            F_AND_2.OUT TO E_SWITCH_2.G;
            MagazinOut.RD_1 TO BOOL2BOOL_2.IN;
            F_AND_1.OUT TO BOOL2BOOL_3.IN;
            PositionSensor TO PUBLISH_0.ID;
            WORD2WORD.OUT TO F_EQ.IN1;
            RobotPosition TO WORD2WORD.IN;
            PresetPosition TO F_EQ.IN2;
          END_CONNECTIONS
        END_SUBAPPLICATION
        EVENT_CONNECTIONS
          SUBSCRIBE_3.INITO TO PUBLISH_2.INIT;
          SUBSCRIBE_3.IND TO WORD2WORD.REQ;
          WORD2WORD.CNF TO E_DELAY_1.START;
          E_DELAY_1.EO TO E_DELAY_1.STOP;
          E_DELAY_1.EO TO PUBLISH_2.REQ;
          INIT TO SUBSCRIBE_3.INIT;
          INIT TO RobotStorageSensorInterlock_1.INIT;
          INIT TO RobotStorageSensorInterlock_2.INIT;
          INIT TO RobotStorageSensorInterlock_3.INIT;
          INIT TO RobotCurrentPosition.INIT;
          RobotCurrentPosition.IND TO WORD2WORD_1.REQ;
          WORD2WORD_1.CNF TO RobotStorageSensorInterlock_1.REQ;
          WORD2WORD_1.CNF TO RobotStorageSensorInterlock_2.REQ;
          WORD2WORD_1.CNF TO RobotStorageSensorInterlock_3.REQ;
          RobotCurrentPosition.INITO TO RobotStorageSensorInterlock.INIT;
          WORD2WORD_1.CNF TO RobotStorageSensorInterlock.REQ;
        END_CONNECTIONS
        DATA_CONNECTIONS
          SUBSCRIBE_3.RD_1 TO WORD2WORD.IN;
          WORD2WORD.OUT TO PUBLISH_2.SD_1;
          RobotCurrentPosition.RD_1 TO WORD2WORD_1.IN;
          WORD2WORD_1.OUT TO RobotStorageSensorInterlock.RobotPosition;
          WORD2WORD_1.OUT TO RobotStorageSensorInterlock_1.RobotPosition;
          WORD2WORD_1.OUT TO RobotStorageSensorInterlock_2.RobotPosition;
          WORD2WORD_1.OUT TO RobotStorageSensorInterlock_3.RobotPosition;
        END_CONNECTIONS
      END_SUBAPPLICATION
      SUBAPPLICATION Robot_OPCUA
        EVENT_INPUT
          INIT;
          REQ;
        END_EVENT
        EVENT_OUTPUT
          CNF;
        END_EVENT
        VAR_INPUT
          CurrentPos : WORD;
        END_VAR
        VAR_OUTPUT
          PostionSp : WORD;
        END_VAR
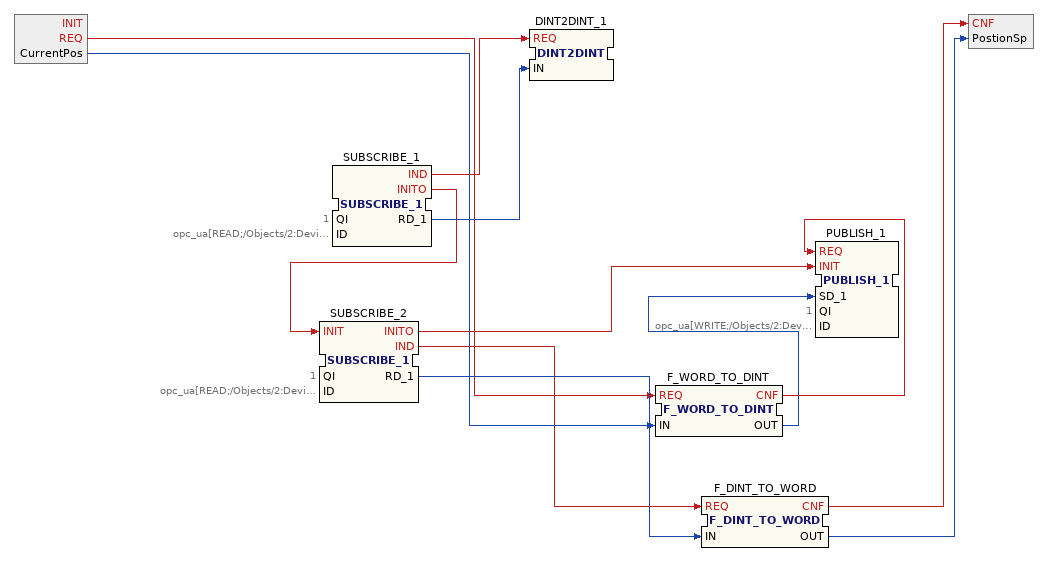
        FBS
          DINT2DINT_1 : DINT2DINT;
          F_WORD_TO_DINT : F_WORD_TO_DINT;
          SUBSCRIBE_2 : SUBSCRIBE_1(QI := 1, ID := opc_ua[READ;/Objects/2:DeviceSet/6:MotionDeviceSystem/5:ProcessData/6:VDMAINVARIABLES/6:SKILL_NMBR]);
          SUBSCRIBE_1 : SUBSCRIBE_1(QI := 1, ID := opc_ua[READ;/Objects/2:DeviceSet/6:MotionDeviceSystem/5:ProcessData/6:VDMAINVARIABLES/6:SKILL_CNTRL]);
          F_DINT_TO_WORD : F_DINT_TO_WORD;
          PUBLISH_1 : PUBLISH_1(QI := 1, ID := opc_ua[WRITE;/Objects/2:DeviceSet/6:MotionDeviceSystem/5:ProcessData/6:VDMAOUTVARIABLES/6:CURRENT_POSITION]);
        END_FBS
        EVENT_CONNECTIONS
          SUBSCRIBE_1.IND TO DINT2DINT_1.REQ;
          F_WORD_TO_DINT.CNF TO PUBLISH_1.REQ;
          SUBSCRIBE_1.INITO TO SUBSCRIBE_2.INIT;
          SUBSCRIBE_2.INITO TO PUBLISH_1.INIT;
          SUBSCRIBE_2.IND TO F_DINT_TO_WORD.REQ;
          REQ TO F_WORD_TO_DINT.REQ;
          F_DINT_TO_WORD.CNF TO CNF;
        END_CONNECTIONS
        DATA_CONNECTIONS
          SUBSCRIBE_1.RD_1 TO DINT2DINT_1.IN;
          F_WORD_TO_DINT.OUT TO PUBLISH_1.SD_1;
          SUBSCRIBE_2.RD_1 TO F_DINT_TO_WORD.IN;
          CurrentPos TO F_WORD_TO_DINT.IN;
          F_DINT_TO_WORD.OUT TO PostionSp;
        END_CONNECTIONS
      END_SUBAPPLICATION
      SUBAPPLICATION Robot_IOs
        EVENT_INPUT
          INIT;
          REQ;
        END_EVENT
        EVENT_OUTPUT
          CNF;
        END_EVENT
        VAR_INPUT
          PositionSP : WORD;
        END_VAR
        VAR_OUTPUT
          CurrentPos : WORD;
        END_VAR
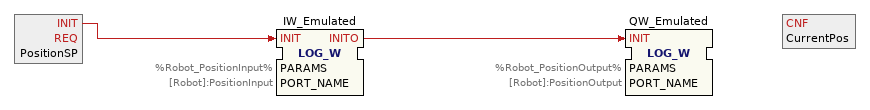
        FBS
          IW_Emulated : LOG_W(PARAMS := %Robot_PositionInput%, PORT_NAME := [Robot]:PositionInput);
          QW_Emulated : LOG_W(PARAMS := %Robot_PositionOutput%, PORT_NAME := [Robot]:PositionOutput);
        END_FBS
        EVENT_CONNECTIONS
          INIT TO IW_Emulated.INIT;
          IW_Emulated.INITO TO QW_Emulated.INIT;
        END_CONNECTIONS
      END_SUBAPPLICATION
      EVENT_CONNECTIONS
        INIT TO Robot_OPCUA.INIT;
        Robot_OPCUA.CNF TO Robot_IOs.REQ;
        INIT TO Robot_IOs.INIT;
        Robot_IOs.CNF TO Robot_OPCUA.REQ;
        INIT TO IO_Logic.INIT;
      END_CONNECTIONS
      DATA_CONNECTIONS
        Robot_OPCUA.PostionSp TO Robot_IOs.PositionSP;
        Robot_IOs.CurrentPos TO Robot_OPCUA.CurrentPos;
      END_CONNECTIONS
    END_SUBAPPLICATION
    SUBAPPLICATION InnerTable
      EVENT_INPUT
        INIT;
      END_EVENT
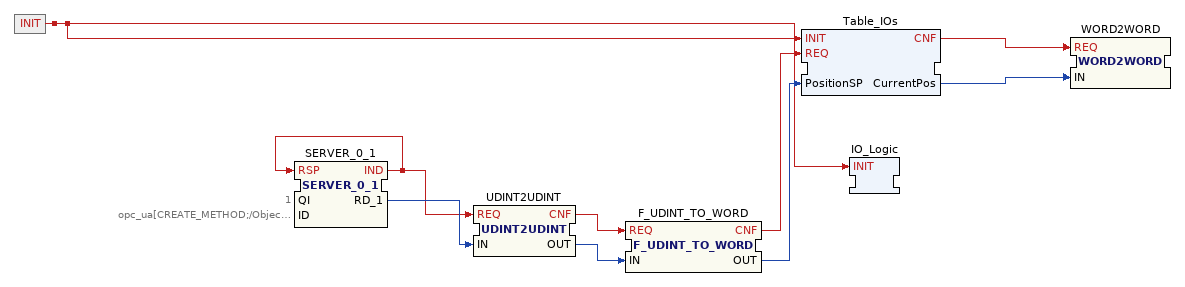
      FBS
        SERVER_0_1 : SERVER_0_1(QI := 1, ID := opc_ua[CREATE_METHOD;/Objects/7:WeissAxis/7:AxisSkillManager/7:MC_MovePresetPosition/7:SetStartParameter]);
        UDINT2UDINT : UDINT2UDINT;
        F_UDINT_TO_WORD : F_UDINT_TO_WORD;
        WORD2WORD : WORD2WORD;
      END_FBS
      SUBAPPLICATION IO_Logic
        EVENT_INPUT
          INIT;
        END_EVENT
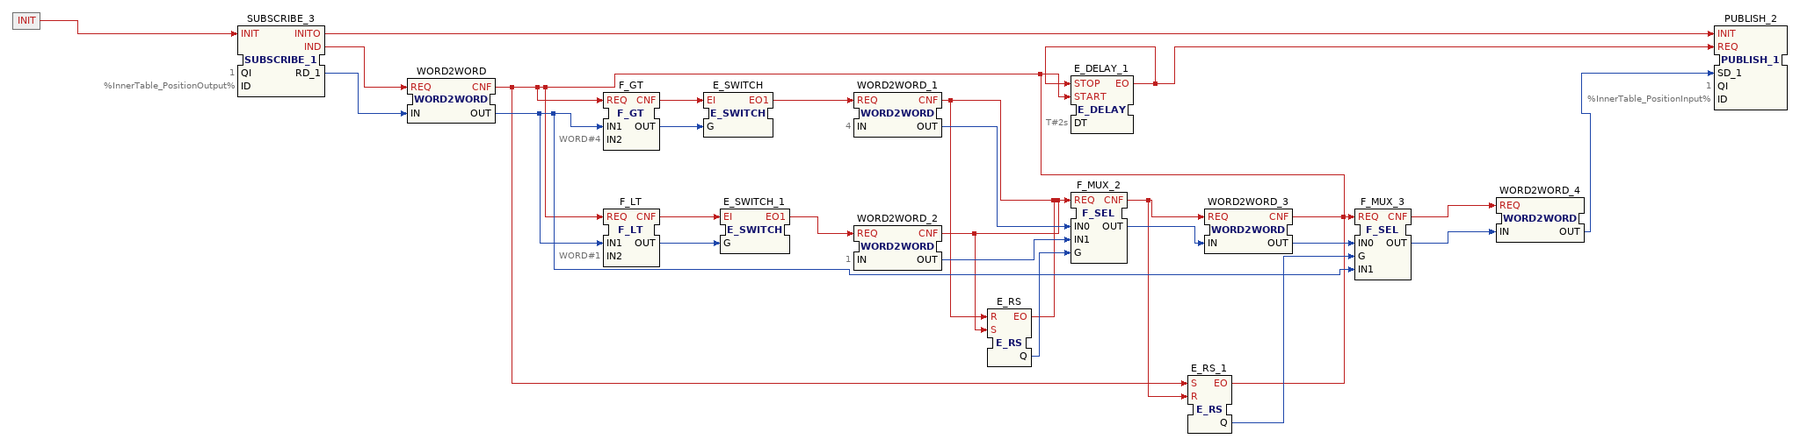
        FBS
          SUBSCRIBE_3 : SUBSCRIBE_1(QI := 1, ID := %InnerTable_PositionOutput%);
          WORD2WORD : WORD2WORD;
          E_DELAY_1 : E_DELAY(DT := T#2s);
          PUBLISH_2 : PUBLISH_1(QI := 1, ID := %InnerTable_PositionInput%);
          F_GT : F_GT(IN2 := WORD#4);
          F_LT : F_LT(IN2 := WORD#1);
          WORD2WORD_1 : WORD2WORD(IN := 4);
          WORD2WORD_2 : WORD2WORD(IN := 1);
          E_SWITCH : E_SWITCH;
          E_SWITCH_1 : E_SWITCH;
          WORD2WORD_3 : WORD2WORD;
          F_MUX_2 : F_SEL;
          F_MUX_3 : F_SEL;
          E_RS : E_RS;
          E_RS_1 : E_RS;
          WORD2WORD_4 : WORD2WORD;
        END_FBS
        EVENT_CONNECTIONS
          SUBSCRIBE_3.INITO TO PUBLISH_2.INIT;
          SUBSCRIBE_3.IND TO WORD2WORD.REQ;
          E_DELAY_1.EO TO E_DELAY_1.STOP;
          E_DELAY_1.EO TO PUBLISH_2.REQ;
          INIT TO SUBSCRIBE_3.INIT;
          WORD2WORD.CNF TO F_GT.REQ;
          WORD2WORD.CNF TO F_LT.REQ;
          F_GT.CNF TO E_SWITCH.EI;
          E_SWITCH.EO1 TO WORD2WORD_1.REQ;
          F_LT.CNF TO E_SWITCH_1.EI;
          E_SWITCH_1.EO1 TO WORD2WORD_2.REQ;
          WORD2WORD.CNF TO E_DELAY_1.START;
          WORD2WORD_1.CNF TO F_MUX_2.REQ;
          WORD2WORD_2.CNF TO F_MUX_2.REQ;
          F_MUX_2.CNF TO WORD2WORD_3.REQ;
          WORD2WORD_3.CNF TO F_MUX_3.REQ;
          WORD2WORD_1.CNF TO E_RS.R;
          WORD2WORD_2.CNF TO E_RS.S;
          E_RS.EO TO F_MUX_2.REQ;
          WORD2WORD.CNF TO E_RS_1.S;
          F_MUX_2.CNF TO E_RS_1.R;
          E_RS_1.EO TO F_MUX_3.REQ;
          F_MUX_3.CNF TO WORD2WORD_4.REQ;
          WORD2WORD.CNF TO F_MUX_3.REQ;
        END_CONNECTIONS
        DATA_CONNECTIONS
          SUBSCRIBE_3.RD_1 TO WORD2WORD.IN;
          WORD2WORD.OUT TO F_LT.IN1;
          WORD2WORD.OUT TO F_GT.IN1;
          F_GT.OUT TO E_SWITCH.G;
          F_LT.OUT TO E_SWITCH_1.G;
          F_MUX_2.OUT TO WORD2WORD_3.IN;
          WORD2WORD_1.OUT TO F_MUX_2.IN0;
          WORD2WORD_2.OUT TO F_MUX_2.IN1;
          WORD2WORD_3.OUT TO F_MUX_3.IN0;
          E_RS.Q TO F_MUX_2.G;
          E_RS_1.Q TO F_MUX_3.G;
          WORD2WORD.OUT TO F_MUX_3.IN1;
          F_MUX_3.OUT TO WORD2WORD_4.IN;
          WORD2WORD_4.OUT TO PUBLISH_2.SD_1;
        END_CONNECTIONS
      END_SUBAPPLICATION
      SUBAPPLICATION Table_IOs
        EVENT_INPUT
          INIT;
          REQ;
        END_EVENT
        EVENT_OUTPUT
          CNF;
        END_EVENT
        VAR_INPUT
          PositionSP : WORD;
        END_VAR
        VAR_OUTPUT
          CurrentPos : WORD;
        END_VAR
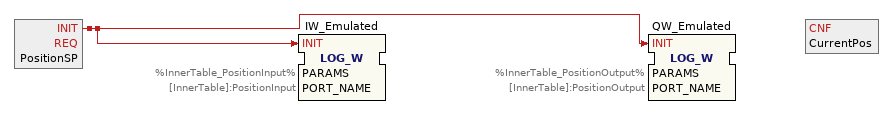
        FBS
          IW_Emulated : LOG_W(PARAMS := %InnerTable_PositionInput%, PORT_NAME := [InnerTable]:PositionInput);
          QW_Emulated : LOG_W(PARAMS := %InnerTable_PositionOutput%, PORT_NAME := [InnerTable]:PositionOutput);
        END_FBS
        EVENT_CONNECTIONS
          INIT TO IW_Emulated.INIT;
          INIT TO QW_Emulated.INIT;
        END_CONNECTIONS
      END_SUBAPPLICATION
      EVENT_CONNECTIONS
        SERVER_0_1.IND TO UDINT2UDINT.REQ;
        INIT TO Table_IOs.INIT;
        INIT TO IO_Logic.INIT;
        UDINT2UDINT.CNF TO F_UDINT_TO_WORD.REQ;
        F_UDINT_TO_WORD.CNF TO Table_IOs.REQ;
        Table_IOs.CNF TO WORD2WORD.REQ;
        SERVER_0_1.IND TO SERVER_0_1.RSP;
      END_CONNECTIONS
      DATA_CONNECTIONS
        SERVER_0_1.RD_1 TO UDINT2UDINT.IN;
        UDINT2UDINT.OUT TO F_UDINT_TO_WORD.IN;
        F_UDINT_TO_WORD.OUT TO Table_IOs.PositionSP;
        Table_IOs.CurrentPos TO WORD2WORD.IN;
      END_CONNECTIONS
    END_SUBAPPLICATION
    SUBAPPLICATION Storage
      EVENT_INPUT
        INIT;
      END_EVENT
